
// ===== library: MasterCopy "GP Drive Control Block" =====

FUNCTION_BLOCK "GP Drive Control Block"   // FB3, STL
{ S7_Optimized_Access := 'FALSE' }
VERSION : 0.1
BEGIN

REGION Network 1
         SET;  // SET RLO=1
         SAVE;  // Save RLO to BR for ENO reset
         L     #Drive_Instance;  // Load the drive instance (sequence within FB call)
         L     0;  // Load 0 into ACCU1 for comparison
         <=I;  // Compare Drive instance to 0 for validation.  instance <=1 causes a jump to label "EXIT"
         JC    EXIT;  // Jump to EXIT routine if drive instance number is <= 0
         TAK;  // Swap ACCU1 and ACCU2 in preparation for calculating offset
         L     1;  // Load one to correct drive instance calculation
         -I;  // Reduce drive insatnce number by for correct offset
         L     16;  // Load 16, the number of bytes in drive data set
         *I;  // Calculate starting byte address for drive instance data within DB
         ITD;  // Convert to 32 bit integer
         SLD   3;  // Shift left three bits to convert to "pointer" construct
         LAR1;  // Load content of ACCU1 in pointer construct to Address Register 1
         L     DIW[AR1, P#0.0];  // Load the SpeedSetpoint input variable (offset +0) into ACCU1
         T     DIW[AR1, P#10.0];  // Transfer contents of ACCU1 (SpeedSetpoint) to Spped_Command output variable (offset +10)
         L     DIW[AR1, P#4.0];  // Load drive status word Status_Word input variable (offset + 4) into ACCU1
         T     DIW[AR1, P#14.0];  // Transfer contents of ACCU1 (Status_Word) to Status Bit Output variables (offset + 14)
         L     DIW[AR1, P#6.0];  // Load the bits that comprise the input Command Word bits (offset + 6) into ACCU1
         CAW;  // Changes the order ofthe bytes within the word in ACCU1 to match order of bytes required by drive
         T     DIW[AR1, P#12.0];  // Tranfer contents of ACCU1 to the Command_Word word output variable (offset + 12)
         SET;  // Set the RLO=1
         SAVE;  // Save the RLO=1 roto the BR bit to turn ENO on
         BE;  // Block End - exit the routine
   EXIT: CLR;  // Clear the RLO (Set to 0)
         SAVE;  // Save RLO to the BR bit, turning off ENO due to error in drive instance number
         BE;  // Block end - exit the routine
END_REGION
END_FUNCTION_BLOCK

// ===== library: MasterCopy "KP8 Tags" =====

VAR_GLOBAL   // PLC tag table "KP8 Tags"
   "Jog_Reverse_Green_KP8" AT %Q51.5 : Bool;   // KP8
   "Enable_Disable_KP8" AT %I50.7 : Bool;   // KP8
   "Drive_Start_KP8" AT %I50.6 : Bool;   // KP8
   "Jog_Reverse_KP8" AT %I50.5 : Bool;   // KP8
   "Switch1_KP8" AT %I50.4 : Bool;   // KP8
   "Enable_Disable_Green_KP8" AT %Q51.7 : Bool;   // KP8
   "Drive_Start_Red_KP8" AT %Q50.6 : Bool;   // KP8
   "Jog_Reverse_Red_KP8" AT %Q50.5 : Bool;   // KP8
   "Switch1_Red_KP8" AT %Q50.4 : Bool;   // KP8
   "RESET_KP8" AT %I50.3 : Bool;   // KP8
   "Drive_Stop_KP8" AT %I50.2 : Bool;   // KP8
   "Jog_Forward_KP8" AT %I50.1 : Bool;   // KP8
   "RESET_Red_KP8" AT %Q50.3 : Bool;   // KP8
   "Drive_Stop_Red_KP8" AT %Q50.2 : Bool;   // KP8
   "Jog_Forward_Red_KP8" AT %Q50.1 : Bool;   // KP8
   "Switch2_KP8" AT %I50.0 : Bool;   // KP8
   "Switch2_Red_KP8" AT %Q50.0 : Bool;   // KP8
   "Enable_Disable_Red_KP8" AT %Q50.7 : Bool;   // KP8
   "Drive_Start_Green_KP8" AT %Q51.6 : Bool;   // KP8
   "Switch1_Green_KP8" AT %Q51.4 : Bool;   // KP8
   "RESET_Green_KP8" AT %Q51.3 : Bool;   // KP8
   "Drive_Stop_Green_KP8" AT %Q51.2 : Bool;   // KP8
   "Jog_Forward_Green_KP8" AT %Q51.1 : Bool;   // KP8
   "Switch2_Green_KP8" AT %Q51.0 : Bool;   // KP8
   "Switch2_Blue_KP8" AT %Q52.0 : Bool;   // KP8
   "Jog_Forward_Blue_KP8" AT %Q52.1 : Bool;   // KP8
   "Drive_Stop_Blue_KP8" AT %Q52.2 : Bool;   // KP8
   "RESET_Blue_KP8" AT %Q52.3 : Bool;   // KP8
   "Switch1_Blue_KP8" AT %Q52.4 : Bool;   // KP8
   "Jog_Reverse_Blue_KP8" AT %Q52.5 : Bool;   // KP8
   "Drive_Start_Blue_KP8" AT %Q52.6 : Bool;   // KP8
   "Enable_Disable_Blue_KP8" AT %Q52.7 : Bool;   // KP8
   "KP8_Red" AT %QB50 : Byte;   // KP8
   "KP8_Green" AT %QB51 : Byte;   // KP8
   "KP8_Blue" AT %QB52 : Byte;   // KP8
END_VAR